// Mitsubishi GX Developer project: 彩灯追灯控制系统   PLC: FX3U

PROGRAM MAIN
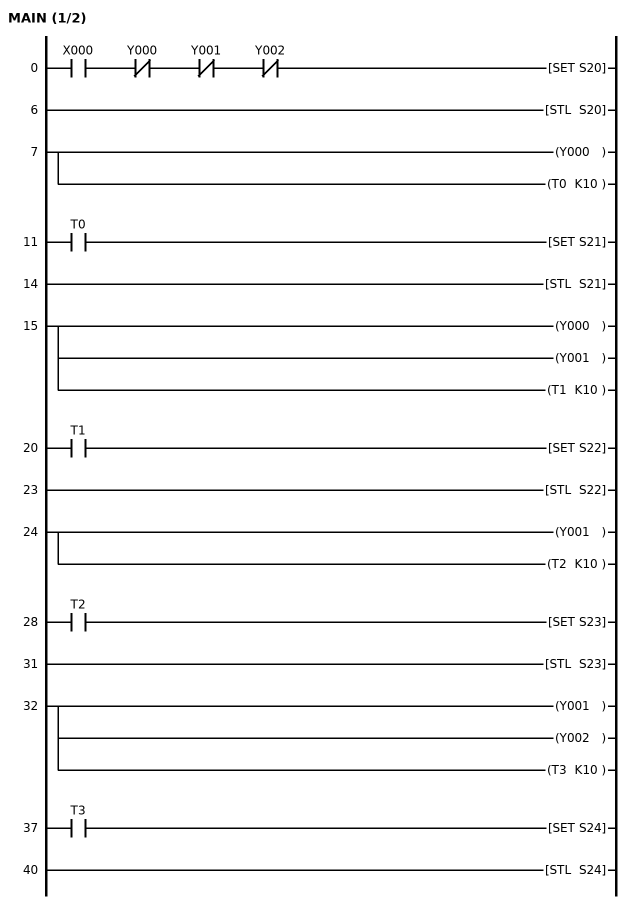
0     LD      X000
      ANI     Y000
      ANI     Y001
      ANI     Y002
      SET     S20
6     STL     S20
7     OUT     Y000
      OUT     T0 K10
11    LD      T0
      SET     S21
14    STL     S21
15    OUT     Y000
      OUT     Y001
      OUT     T1 K10
20    LD      T1
      SET     S22
23    STL     S22
24    OUT     Y001
      OUT     T2 K10
28    LD      T2
      SET     S23
31    STL     S23
32    OUT     Y001
      OUT     Y002
      OUT     T3 K10
37    LD      T3
      SET     S24
40    STL     S24
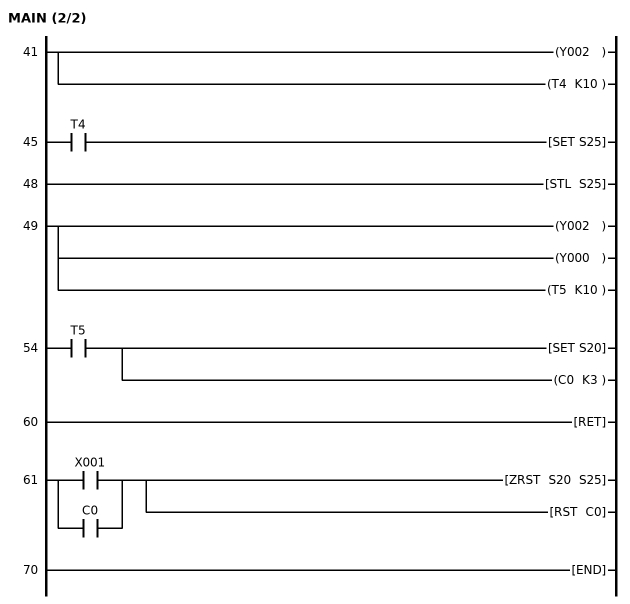
41    OUT     Y002
      OUT     T4 K10
45    LD      T4
      SET     S25
48    STL     S25
49    OUT     Y002
      OUT     Y000
      OUT     T5 K10
54    LD      T5
      SET     S20
      OUT     C0 K3
60    RET
61    LD      X001
      OR      C0
      ZRST    S20 S25
      RST     C0
70    END
END_PROGRAM
